FUNCTION_BLOCK ASR_2EVENTS_TO_SR (* Composite FB for convert 2 EVENTS to ASR *)
  (* Standard: 61499-2; Description: Copyright (c) 2024 HR Agrartechnik GmbH This program and the accompanying materials are made available under the terms of the Eclipse Public License 2.0 which is available at https://www.eclipse.org/legal/epl-2.0/ SPDX-License-Identifier: EPL-2.0 *)
  (* Version 1.0, 2024-04-24, Franz Höpfinger, HR Agrartechnik GmbH *)
  PACKAGE adapter::conversion::unidirectional;
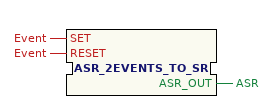
  EVENT_INPUT
    SET; (* Set / Switch on *)
    RESET; (* Reset / Switch off *)
  END_EVENT
  PLUGS
    ASR_OUT : adapter::types::unidirectional::ASR; (* Adapter Output *)
  END_PLUGS
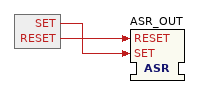
  EVENT_CONNECTIONS
    RESET TO ASR_OUT.RESET;
    SET TO ASR_OUT.SET;
  END_CONNECTIONS
END_FUNCTION_BLOCK
